PROGRAM MAIN
VAR
	bEnable : BOOL; 
	bStart : BOOL; 
END_VAR

bEnable := bStart;

END_PROGRAM

(* stored: Version 1.1.0.1, ProductVersion 3.1.4024.12
   POU MAIN: Id {4050dae3-d7dc-4ead-9eb6-5b390007f3e7}, SpecialFunc None *)
